PROGRAM PROG //Place to program application specific code
VAR
	
END_VAR

END_PROGRAM

(* stored: Version 1.1.0.1, ProductVersion 3.1.4024.5
   POU PROG: Id {971c9f67-c7aa-4c3b-a151-6b6f987c9db5}, SpecialFunc None *)
